TYPE
    ST_SetupMotor :
    STRUCT
		//A倉軌道
        WareHouseCV_10          : ST_MotorPara;
        WareHouseCV_09          : ST_MotorPara;
        WareHouseCV_08          : ST_MotorPara;
        WareHouseCV_07          : ST_MotorPara;
        WareHouseCV_06          : ST_MotorPara;
        WareHouseCV_05          : ST_MotorPara;
        WareHouseCV_04          : ST_MotorPara;
        WareHouseCV_03          : ST_MotorPara;
        WareHouseCV_02          : ST_MotorPara;
        WareHouseCV_01          : ST_MotorPara;
		//B倉軌道
        WareHouseCV_20          : ST_MotorPara;
        WareHouseCV_19          : ST_MotorPara;
        WareHouseCV_18          : ST_MotorPara;
        WareHouseCV_17          : ST_MotorPara;
        WareHouseCV_16          : ST_MotorPara;
        WareHouseCV_15          : ST_MotorPara;
        WareHouseCV_14          : ST_MotorPara;
        WareHouseCV_13          : ST_MotorPara;
        WareHouseCV_12          : ST_MotorPara;
        WareHouseCV_11          : ST_MotorPara;
		
        UpCV                    : ST_MotorPara;//上層軌道
		
        LowCV                   : ST_MotorPara;//下層軌道
		
        PullOutCV_A             : ST_MotorPara;//空盒軌道
		
        PullOutCV_B             : ST_MotorPara;//待拔針軌道 
		
        TransmitSameSideCV      : ST_MotorPara;//同尺寸軌道
		
        TransmitDifferentSideCV : ST_MotorPara; //配針軌道
    END_STRUCT
END_TYPE

(* stored: Version 1.1.0.1, ProductVersion 3.1.4024.13
   DUT ST_SetupMotor: Id {66a50f0d-dc50-4170-8474-cb2bc9306d58} *)
